# EPICS autosave request: ADEuresys/iocs/EuresysIOC/iocBoot/iocViewWorks/auto_settings.req
file "Euresys_settings.req",              P=$(P),  R=cam1:
file "NDStdArrays_settings.req",          P=$(P),  R=image1:
file "commonPlugin_settings.req",         P=$(P)
